// SIMATIC S7-200 project (STEP 7-Micro/WIN), CPU 226 REL 01.23

ORGANIZATION_BLOCK MAIN:OB1
TITLE=
BEGIN
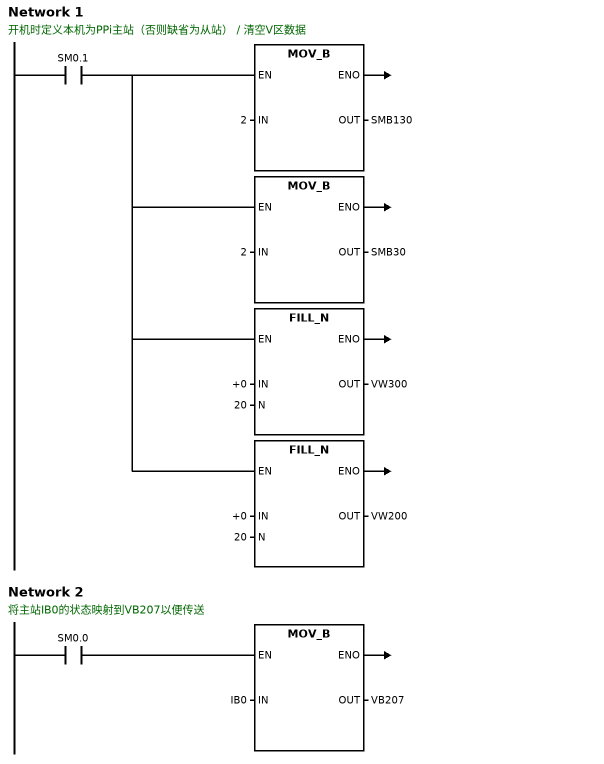
Network 1
// 开机时定义本机为PPi主站（否则缺省为从站）
// 清空V区数据
LD     SM0.1
MOVB   2, SMB130
MOVB   2, SMB30
FILL   +0, VW300, 20
FILL   +0, VW200, 20
Network 2
// 将主站IB0的状态映射到VB207以便传送
LD     SM0.0
MOVB   IB0, VB207
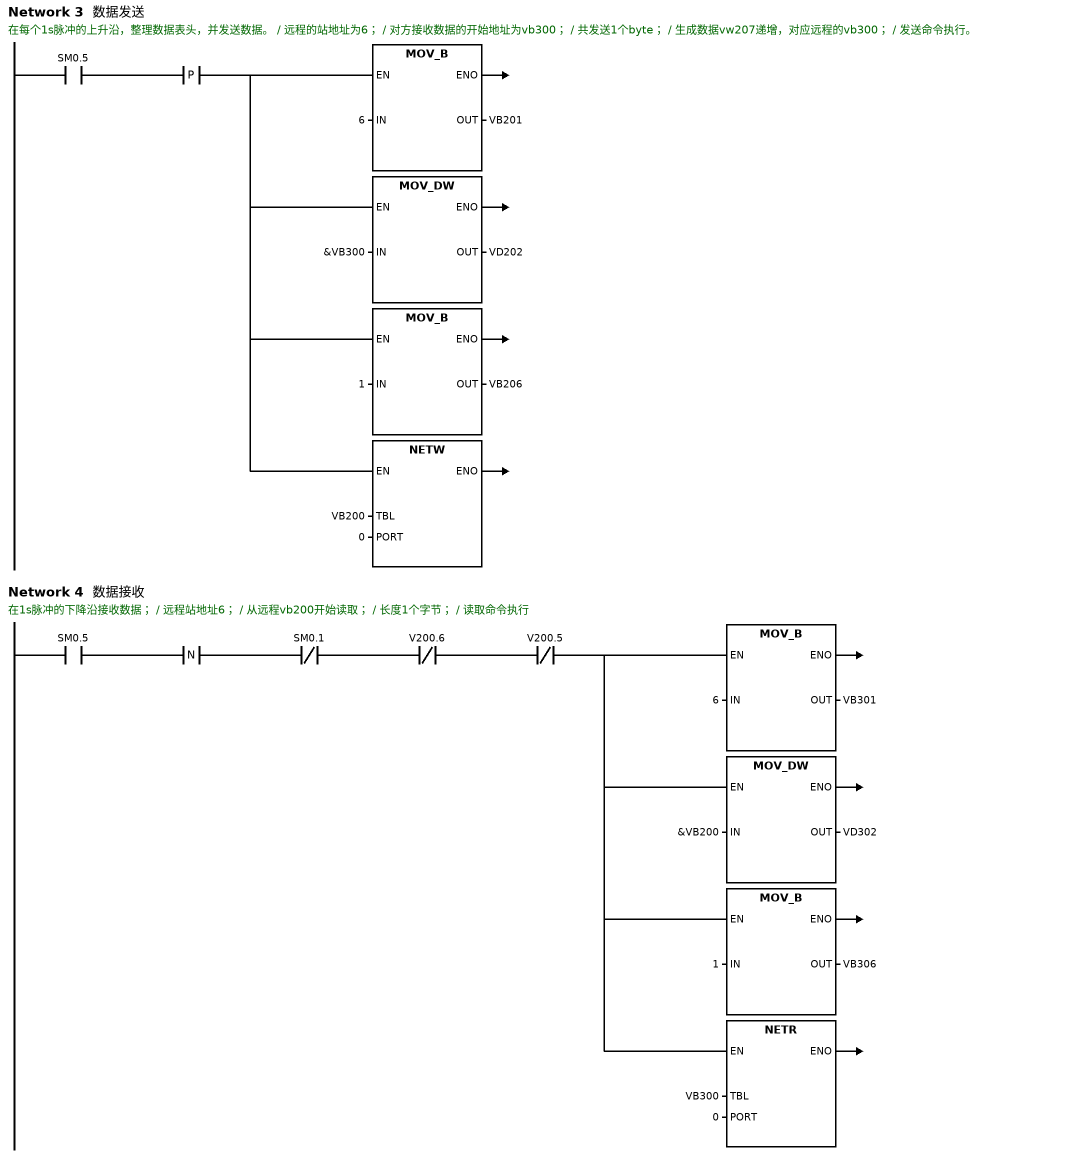
Network 3 // 数据发送
// 在每个1s脉冲的上升沿，整理数据表头，并发送数据。
// 远程的站地址为6；
// 对方接收数据的开始地址为vb300；
// 共发送1个byte；
// 生成数据vw207递增，对应远程的vb300；
// 发送命令执行。
LD     SM0.5
EU
MOVB   6, VB201
MOVD   &VB300, VD202
MOVB   1, VB206
?233   VB200, 0
Network 4 // 数据接收
// 在1s脉冲的下降沿接收数据；
// 远程站地址6；
// 从远程vb200开始读取；
// 长度1个字节；
// 读取命令执行
LD     SM0.5
ED
AN     SM0.1
AN     V200.6
AN     V200.5
MOVB   6, VB301
MOVD   &VB200, VD302
MOVB   1, VB306
?232   VB300, 0
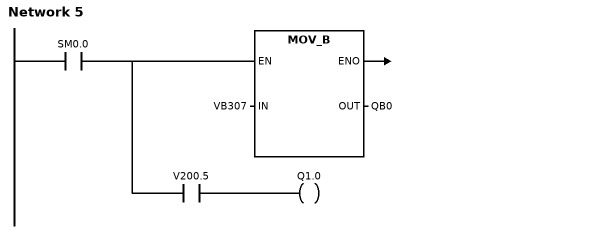
Network 5
LD     SM0.0
MOVB   VB307, QB0
A      V200.5
=      Q1.0
END_ORGANIZATION_BLOCK
